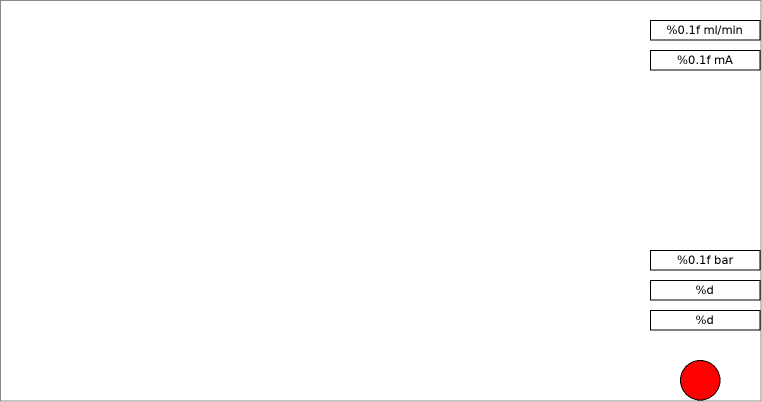
VISUALIZATION Q2  // 762x402
    Rectangle (650,20 110x20), "%0.1f ml/min", text variable: IOs_Variables.Q2_CALCULETED_FLOW
    Rectangle (650,280 110x20), "%d", text variable: LEDS.M2_FB_GetPositionIs.PositionIs
    Rectangle (650,250 110x20), "%0.1f bar", text variable: IOs_Variables.Q2_PRESSURE_SENSOR_VALUE
    Rectangle (650,310 110x20), "%d", text variable: Q2.STEP
    Ellipse (680,360 40x40), colour toggle: (LEDS.M2_FB_GetEnableState.IsEnabled) <> 0
    Rectangle (650,50 110x20), "%0.1f mA", text variable: IOs_Variables.Q2_CURRENT
END_VISUALIZATION

(* stored: Version 1.1.0.1, ProductVersion 3.1.0.26
   Visu Q2: Id {dbd0f5aa-d47c-4aee-82b7-782f2dfe62c6} *)
